// TIA Portal V16 export
// export: Created 2023-08-28T09:37:51.341577Z, ExportSetting WithDefaults, DisplayName Totally Integrated Automation Portal, DisplayVersion V16 Update 6, DisplayName TIA Portal Version Control Interface, DisplayVersion V16 Update 2, DisplayName TIA Portal Openness, DisplayVersion V16 Update 6, DisplayName STEP 7 Professional, DisplayVersion V16 Update 6, DisplayName STEP 7 Safety, DisplayVersion V16, DisplayName WinCC Advanced, DisplayVersion V16 Update 6
DATA_BLOCK "dbTags_master_RTU"   // DB90
TITLE = Master
{ S7_Optimized_Access := 'FALSE' }
AUTHOR : rtecmer
VERSION : 0.1
// Instancja dla funkcji Mdbus RTU komunikacja z masterem MT101
// stored: AutoNumber false, DBAccessibleFromOPCUA true, IsOnlyStoredInLoadMemory false, IsWriteProtectedInAS false
   VAR
      "step" : USInt := 1;
      edge : Bool := false;
      modbusCommLoad { S7_SetPoint := 'True'} : "typeModbusCommLoad";
      modbusMaster { S7_SetPoint := 'True'} : "typeModbusSlave";
   END_VAR
BEGIN
END_DATA_BLOCK
